Staubli VAL3: exeBlink.pgx

program exeBlink(dio x_dDio, num x_nInterval)
begin

  while true

    x_dDio=true
    delay(x_nInterval)
    x_dDio=false
    delay(x_nInterval)

  endWhile

end
